// TIA Portal V20 export
DATA_BLOCK "SP204"   // DB315
// stored: MemoryReserve 100
   VAR
      "MAIN OP EMERGENCY STOP CH.A" : Bool;
      SPARE : Bool;
      SPARE_1 : Bool;
      SPARE_2 : Bool;
      "MAIN OP EMERGENCY STOP CH.B" : Bool;
      SPARE_3 : Bool;
      SPARE_4 : Bool;
      SPARE_5 : Bool;
   END_VAR
BEGIN
END_DATA_BLOCK
